Fanuc KAREL source: kt00747.KL

-- PROVISIONAL review KL for V940-1; original PC SHA256 698252181dbf59b6e03094fe70870f8cd41080b390be0b213c8d9cdaca4c6788
-- Incomplete behavior may be omitted. Consult companion uncertainty JSON. Do not deploy.
PROGRAM KT00747
%NOLOCKGROUP
BEGIN
  -- V9_ZERO_TABLE_METADATA_HINT layout=0001; no indexed target words; source/name/runtime held
  -- UNRESOLVED_PC offsets 5-18; opcodes 22,1D,23
  -- UNRESOLVED_PC offsets 23-27; opcodes 7F
END KT00747
